TYPE T_CodeURL : STRING[20];
END_TYPE

(* stored: Version 1.1.0.1
   DUT T_CodeURL: Id {1d93f398-db04-4c7f-834e-42f4abb88668} *)
